// TIA Portal V15.1 export
// export: Created 2024-06-21T08:41:14.0911961Z, ExportSetting WithDefaults, DisplayName Totally Integrated Automation Portal, DisplayVersion V15.1 Update 5, DisplayName TIA Portal Openness, DisplayVersion V15.1 Update 5, DisplayName SINAMICS Startdrive Advanced, DisplayVersion V15.1, DisplayName G130, G150, S120, S150, SINAMICS MV, S210, DisplayVersion V15.1, DisplayName G110M, G120, G120C, G120D, G120P, DisplayVersion V15.1, DisplayName STEP 7 Professional, DisplayVersion V15.1 Update 5, DisplayName STEP 7 Safety, DisplayVersion V15.1, DisplayName WinCC Professional, DisplayVersion V15.1 Update 5, DisplayName SIMATIC Visualization Architect, DisplayVersion V15.1
FUNCTION_BLOCK "LGBSickDL100"   // FB6673, FBD
TITLE = LSickDL100 / LGBSickDL100
{ S7_Optimized_Access := 'TRUE' }
VERSION : 0.1
// LSickDL100 / LGBSickDL100
// stored: AutoNumber false, IsIECCheckEnabled false, IsRetainMemResEnabled false, MemoryReserve 100, SetENOAutomatically False, UDAEnableTagReadback false
   VAR_INPUT
      I_TEL_M04_Inputs { ExternalAccessible := 'False'; ExternalVisible := 'False'; ExternalWritable := 'False'} : "Sick_TEL_M04_Inputs";   // Sick input module M04
      I_TEL_M10_Inputs { ExternalAccessible := 'False'; ExternalVisible := 'False'; ExternalWritable := 'False'} : "Sick_TEL_M10_Inputs";   // Sick input module M10
      I_TEL_M13_Inputs_P1 { ExternalAccessible := 'False'; ExternalVisible := 'False'; ExternalWritable := 'False'} : "Sick_TEL_M13_Inputs_Part_1";   // Sick input module M13 part 1
      I_TEL_M13_Inputs_P2 { ExternalAccessible := 'False'; ExternalVisible := 'False'; ExternalWritable := 'False'} : "Sick_TEL_M13_Inputs_Part_2";   // Sick input module M13 part 2
      I_TurnLaserOff { ExternalAccessible := 'False'; ExternalVisible := 'False'; ExternalWritable := 'False'} : Bool;   // Turn laser off, this will cause a alarm B !
      C_ReceptionQualityMin { ExternalAccessible := 'False'; ExternalVisible := 'False'; ExternalWritable := 'False'} : Int := -96;   // Minimum reception quality level before alarm C
   END_VAR
   VAR_OUTPUT
      O_TEL_M10_Outputs { ExternalAccessible := 'False'; ExternalVisible := 'False'; ExternalWritable := 'False'} : "Sick_TEL_M10_Outputs";   // Sick output module M10
      O_Distance { ExternalAccessible := 'False'; ExternalVisible := 'False'; ExternalWritable := 'False'} : DInt;   // Current distance in the current resolution under consideration of offset. Depending on resolution, one digit corresponds to 0.1 to 100 mm.
      O_Speed { ExternalAccessible := 'False'; ExternalVisible := 'False'; ExternalWritable := 'False'} : DInt;   // Current speed in selected resolution. Depending on resolution, one digit corresponds to 0.1m/s to 100 mm/s.
      O_DeviceTemp { ExternalAccessible := 'False'; ExternalVisible := 'False'; ExternalWritable := 'False'} : SInt := 0;   // Device temperature [°C]
      O_ReceptionQuality { ExternalAccessible := 'False'; ExternalVisible := 'False'; ExternalWritable := 'False'} : Int := 0;   // Device-specific value for the signal reception quality
      O_OperatingHours { ExternalAccessible := 'False'; ExternalVisible := 'False'; ExternalWritable := 'False'} : Int := 0;   // Operating hours in 10 hour units.
      O_LaserOff { ExternalAccessible := 'False'; ExternalVisible := 'False'; ExternalWritable := 'False'} : Bool;   // Laser is off
      O_AlarmABCondition { ExternalAccessible := 'False'; ExternalVisible := 'False'; ExternalWritable := 'False'} : Bool;   // Alarm AB Condition
      O_AlarmA { ExternalAccessible := 'False'; ExternalVisible := 'False'; ExternalWritable := 'False'} : Bool;   // Alarm A
      O_AlarmB { ExternalAccessible := 'False'; ExternalVisible := 'False'; ExternalWritable := 'False'} : Bool;   // Alarm B
      O_AlarmC { ExternalAccessible := 'False'; ExternalVisible := 'False'; ExternalWritable := 'False'} : Bool;   // Alarm C
      O_AlarmD { ExternalAccessible := 'False'; ExternalVisible := 'False'; ExternalWritable := 'False'} : Bool;   // Alarm D
      H_AlarmDWord { ExternalAccessible := 'False'; ExternalVisible := 'False'; ExternalWritable := 'False'} : DWord;   // Alarm Word
   END_VAR
   VAR_IN_OUT
      IO_Modes : "Modes";   // Modes
      H_HMI : "H_HMI";   // Animation
      H_GBSickDL100 : "H_GBSickDL100";   // Animation
   END_VAR
   VAR
      AB_PlausibilityError { ExternalAccessible := 'False'; ExternalVisible := 'False'; ExternalWritable := 'False'} : Bool;   // No valid measurement value can be calculated.
      AB_TemperatureError { ExternalAccessible := 'False'; ExternalVisible := 'False'; ExternalWritable := 'False'} : Bool;   // The device is also operated outside of the specified temperature range
      AB_SignalLevelError { ExternalAccessible := 'False'; ExternalVisible := 'False'; ExternalWritable := 'False'} : Bool;   // The measured signal level is too low.
      AB_LaserError { ExternalAccessible := 'False'; ExternalVisible := 'False'; ExternalWritable := 'False'} : Bool;   // The laser may have reached the end of its service life
      AB_LaserOff { ExternalAccessible := 'False'; ExternalVisible := 'False'; ExternalWritable := 'False'} : Bool;   // Laser is off
      AB_ValueValid { ExternalAccessible := 'False'; ExternalVisible := 'False'; ExternalWritable := 'False'} : Bool;   // 1= No distance or speed measurement value can be read. 0 = Current measurement value is valid
      AC_PlausibilityWarning { ExternalAccessible := 'False'; ExternalVisible := 'False'; ExternalWritable := 'False'} : Bool;   // Measured values are impaired.
      AC_TemperatureWarning { ExternalAccessible := 'False'; ExternalVisible := 'False'; ExternalWritable := 'False'} : Bool;   // The ambient temperature is only just within the permissible range.
      AC_SignalLevelWarning { ExternalAccessible := 'False'; ExternalVisible := 'False'; ExternalWritable := 'False'} : Bool;   // The measured signal level is close to the permissible range.
      AC_LaserWarning { ExternalAccessible := 'False'; ExternalVisible := 'False'; ExternalWritable := 'False'} : Bool;   // The laser has reached its service life.
      AC_ReceptionQuality { ExternalAccessible := 'False'; ExternalVisible := 'False'; ExternalWritable := 'False'} : Bool;   // Device-specific value for the signal reception quality
      AlarmABCondition { ExternalAccessible := 'False'; ExternalVisible := 'False'; ExternalWritable := 'False'} : Bool;   // Alarm AB Condition
      AlarmA { ExternalAccessible := 'False'; ExternalVisible := 'False'; ExternalWritable := 'False'} : Bool;   // Alarm A
      AlarmB { ExternalAccessible := 'False'; ExternalVisible := 'False'; ExternalWritable := 'False'} : Bool;   // Alarm B
      AlarmC { ExternalAccessible := 'False'; ExternalVisible := 'False'; ExternalWritable := 'False'} : Bool;   // Alarm C
      AlarmD { ExternalAccessible := 'False'; ExternalVisible := 'False'; ExternalWritable := 'False'} : Bool;   // Alarm D
   END_VAR
   VAR_TEMP   // added for the SCL form of the ladder/FBD networks
      _w1 : Bool;
   END_VAR
BEGIN

REGION Network 1: **** 2.2 - Alarms - Alarm Generation **** Alarm B laser is turned off
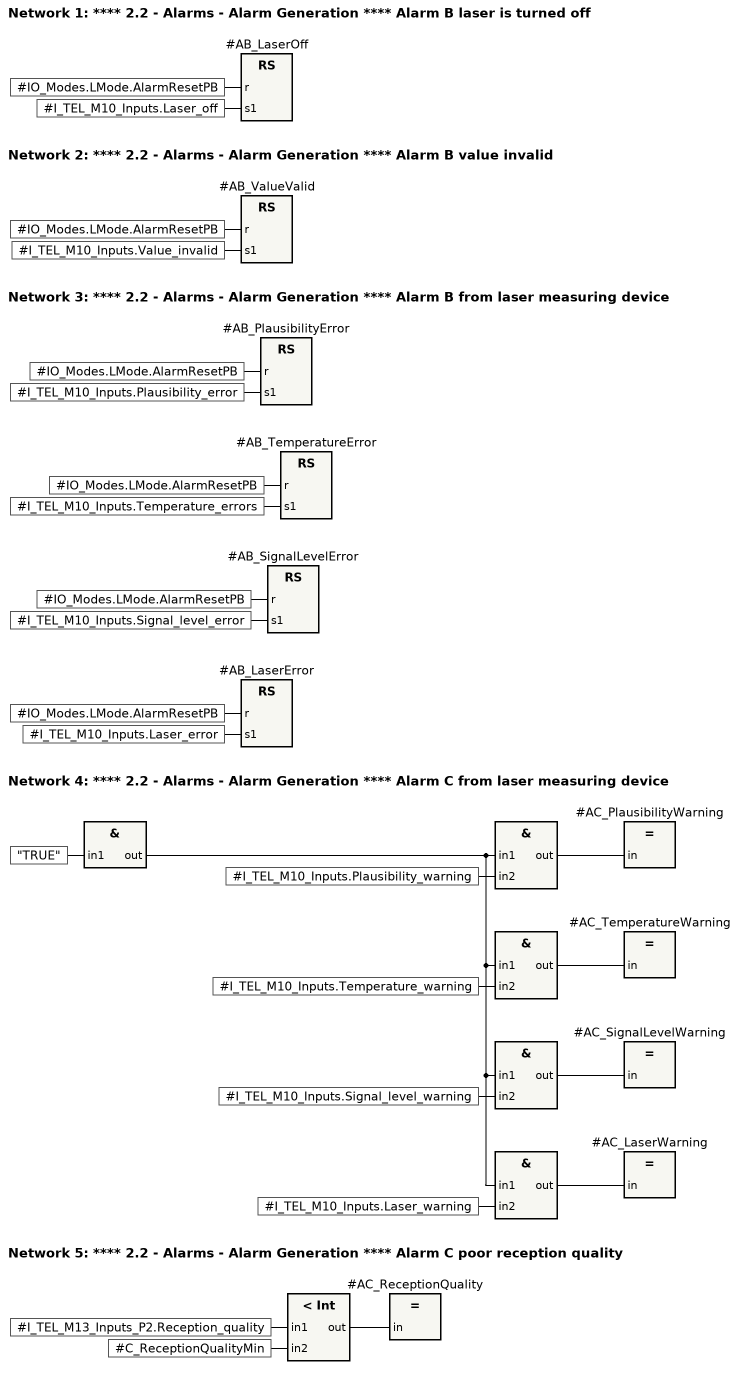
   IF #IO_Modes.LMode.AlarmResetPB THEN
       #AB_LaserOff := FALSE;   // RS flip-flop
   END_IF;
   IF #I_TEL_M10_Inputs.Laser_off THEN #AB_LaserOff := TRUE; END_IF;
END_REGION

REGION Network 2: **** 2.2 - Alarms - Alarm Generation **** Alarm B value invalid
   IF #IO_Modes.LMode.AlarmResetPB THEN
       #AB_ValueValid := FALSE;   // RS flip-flop
   END_IF;
   IF #I_TEL_M10_Inputs.Value_invalid THEN #AB_ValueValid := TRUE; END_IF;
END_REGION

REGION Network 3: **** 2.2 - Alarms - Alarm Generation **** Alarm B from laser measuring device
   IF #IO_Modes.LMode.AlarmResetPB THEN
       #AB_PlausibilityError := FALSE;   // RS flip-flop
   END_IF;
   IF #I_TEL_M10_Inputs.Plausibility_error THEN #AB_PlausibilityError := TRUE; END_IF;
   IF #IO_Modes.LMode.AlarmResetPB THEN
       #AB_TemperatureError := FALSE;   // RS flip-flop: __ 40°C l l l~l 20°C l l l l l l 0°C l l l l -10°C l l (__)
   END_IF;
   IF #I_TEL_M10_Inputs.Temperature_errors THEN #AB_TemperatureError := TRUE; END_IF;
   IF #IO_Modes.LMode.AlarmResetPB THEN
       #AB_SignalLevelError := FALSE;   // RS flip-flop
   END_IF;
   IF #I_TEL_M10_Inputs.Signal_level_error THEN #AB_SignalLevelError := TRUE; END_IF;
   IF #IO_Modes.LMode.AlarmResetPB THEN
       #AB_LaserError := FALSE;   // RS flip-flop
   END_IF;
   IF #I_TEL_M10_Inputs.Laser_error THEN #AB_LaserError := TRUE; END_IF;
END_REGION

REGION Network 4: **** 2.2 - Alarms - Alarm Generation **** Alarm C from laser measuring device
   #AC_PlausibilityWarning := "TRUE" AND #I_TEL_M10_Inputs.Plausibility_warning;
   #AC_TemperatureWarning := "TRUE" AND #I_TEL_M10_Inputs.Temperature_warning;   // __ 40°C l l l~l 20°C l l l l l l 0°C l l l l -10°C l l (__)
   #AC_SignalLevelWarning := "TRUE" AND #I_TEL_M10_Inputs.Signal_level_warning;
   #AC_LaserWarning := "TRUE" AND #I_TEL_M10_Inputs.Laser_warning;
END_REGION

REGION Network 5: **** 2.2 - Alarms - Alarm Generation **** Alarm C poor reception quality
   #AC_ReceptionQuality := #I_TEL_M13_Inputs_P2.Reception_quality < #C_ReceptionQualityMin;   // ^ Reception quality (%) l -32db l_______________ l \ OK area min. l \ if quality drops below this level .setting l---------------------------------------\------------------------------------------------------------- an alarm C is created. l \ alarm C area -96db l________________________\___________________________> Time (h) l This can be caused: -by dirt on the mirror. -misalignment (ex. cuased by moving the mirror). -...
END_REGION

REGION Network 6: **** 4.6 - Machine Status - Indication **** Icon Animation
   // Icon Animation
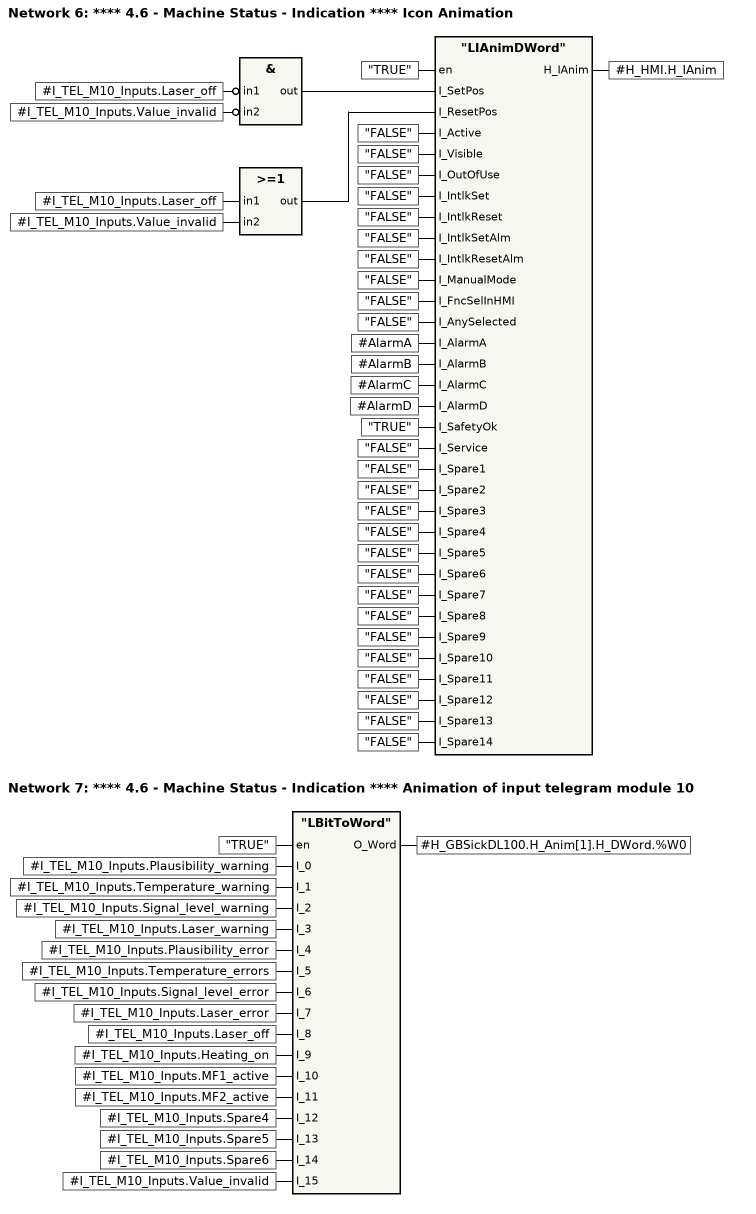
   IF "TRUE" THEN
       "LIAnimDWord"(I_SetPos := NOT #I_TEL_M10_Inputs.Laser_off AND NOT #I_TEL_M10_Inputs.Value_invalid,   // HMI PLC __________________________________________________________ l _SIEMENS____________________________SIMATIC HMI_____ l ___________________ l l l l l_l_l_l______________l l l l l l SIEMENS SIMATIC l l l l l l ________S7-1500 l l l l l l l___________O_l l l l Icon l l l l l l l l ____ l l l l l l l l l l l l l l l l l l l____l <<-------==================l= l========= l l l l l l l l l l______________l l l l IAnim l l l ___ l l l l l l __l l__ l l l l l l l__ __l l l l l l l l___l l l l l l l l l l_____________________________________________________ l l l__________________ l l_________________________________________________________ l Icon animation word is send to the HMI to be used in ex .modezone screen _
                     I_ResetPos := #I_TEL_M10_Inputs.Laser_off OR #I_TEL_M10_Inputs.Value_invalid,
                     I_Active := "FALSE",
                     I_Visible := "FALSE",
                     I_OutOfUse := "FALSE",
                     I_IntlkSet := "FALSE",
                     I_IntlkReset := "FALSE",
                     I_IntlkSetAlm := "FALSE",
                     I_IntlkResetAlm := "FALSE",
                     I_ManualMode := "FALSE",
                     I_FncSelInHMI := "FALSE",
                     I_AnySelected := "FALSE",
                     I_AlarmA := #AlarmA,
                     I_AlarmB := #AlarmB,
                     I_AlarmC := #AlarmC,
                     I_AlarmD := #AlarmD,
                     I_SafetyOk := "TRUE",
                     I_Service := "FALSE",
                     I_Spare1 := "FALSE",
                     I_Spare2 := "FALSE",
                     I_Spare3 := "FALSE",
                     I_Spare4 := "FALSE",
                     I_Spare5 := "FALSE",
                     I_Spare6 := "FALSE",
                     I_Spare7 := "FALSE",
                     I_Spare8 := "FALSE",
                     I_Spare9 := "FALSE",
                     I_Spare10 := "FALSE",
                     I_Spare11 := "FALSE",
                     I_Spare12 := "FALSE",
                     I_Spare13 := "FALSE",
                     I_Spare14 := "FALSE",
                     H_IAnim => #H_HMI.H_IAnim);
   END_IF;
END_REGION

REGION Network 7: **** 4.6 - Machine Status - Indication **** Animation of input telegram module 10
   // Animation
   IF "TRUE" THEN
       "LBitToWord"(I_0 := #I_TEL_M10_Inputs.Plausibility_warning,   // HMI PLC __________________________________________________________ l _SIEMENS____________________________SIMATIC HMI_____ l ___________________ l l l l l_l_l_l______________l l l l l l SIEMENS SIMATIC l l l ________________ l l l ________S7-1500 l l l l_____________ X l l l l l___________O_l l l l l l l l l l l l l l l Popup or l l l l l l l l l l screen. l l l l l l l l l l l <<-------==================l= l========= l l l l l l l Anim l l l l l______________l l l l l_______________l l l l ___ l l l l l l __l l__ l l l l l l l__ __l l l l l l l l___l l l l l l l l l l_____________________________________________________ l l l__________________ l l_________________________________________________________ l Animation word is send to the HMI to be used in object screen or popup _
                    I_1 := #I_TEL_M10_Inputs.Temperature_warning,
                    I_2 := #I_TEL_M10_Inputs.Signal_level_warning,
                    I_3 := #I_TEL_M10_Inputs.Laser_warning,
                    I_4 := #I_TEL_M10_Inputs.Plausibility_error,
                    I_5 := #I_TEL_M10_Inputs.Temperature_errors,
                    I_6 := #I_TEL_M10_Inputs.Signal_level_error,
                    I_7 := #I_TEL_M10_Inputs.Laser_error,
                    I_8 := #I_TEL_M10_Inputs.Laser_off,
                    I_9 := #I_TEL_M10_Inputs.Heating_on,
                    I_10 := #I_TEL_M10_Inputs.MF1_active,
                    I_11 := #I_TEL_M10_Inputs.MF2_active,
                    I_12 := #I_TEL_M10_Inputs.Spare4,
                    I_13 := #I_TEL_M10_Inputs.Spare5,
                    I_14 := #I_TEL_M10_Inputs.Spare6,
                    I_15 := #I_TEL_M10_Inputs.Value_invalid,
                    O_Word => #H_GBSickDL100.H_Anim[1].H_DWord.%W0);
   END_IF;
END_REGION

REGION Network 8: **** 4.6 - Machine Status - Indication **** Animation of output telegram module 10
   // Animation
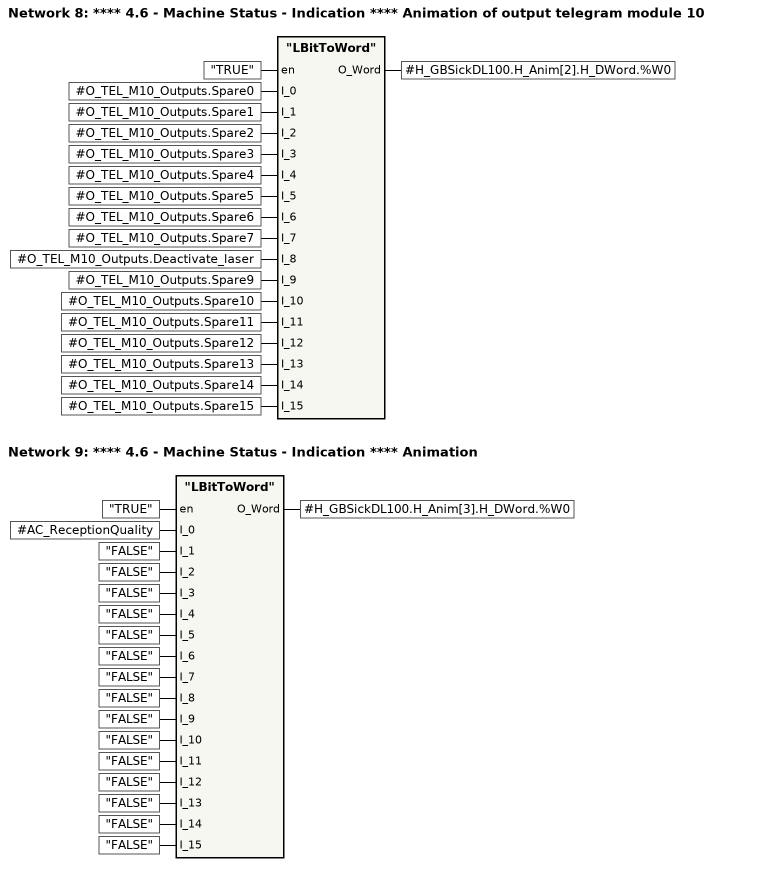
   IF "TRUE" THEN
       "LBitToWord"(I_0 := #O_TEL_M10_Outputs.Spare0,   // HMI PLC __________________________________________________________ l _SIEMENS____________________________SIMATIC HMI_____ l ___________________ l l l l l_l_l_l______________l l l l l l SIEMENS SIMATIC l l l ________________ l l l ________S7-1500 l l l l_____________ X l l l l l___________O_l l l l l l l l l l l l l l l Popup or l l l l l l l l l l screen. l l l l l l l l l l l <<-------==================l= l========= l l l l l l l Anim l l l l l______________l l l l l_______________l l l l ___ l l l l l l __l l__ l l l l l l l__ __l l l l l l l l___l l l l l l l l l l_____________________________________________________ l l l__________________ l l_________________________________________________________ l Animation word is send to the HMI to be used in object screen or popup _
                    I_1 := #O_TEL_M10_Outputs.Spare1,
                    I_2 := #O_TEL_M10_Outputs.Spare2,
                    I_3 := #O_TEL_M10_Outputs.Spare3,
                    I_4 := #O_TEL_M10_Outputs.Spare4,
                    I_5 := #O_TEL_M10_Outputs.Spare5,
                    I_6 := #O_TEL_M10_Outputs.Spare6,
                    I_7 := #O_TEL_M10_Outputs.Spare7,
                    I_8 := #O_TEL_M10_Outputs.Deactivate_laser,
                    I_9 := #O_TEL_M10_Outputs.Spare9,
                    I_10 := #O_TEL_M10_Outputs.Spare10,
                    I_11 := #O_TEL_M10_Outputs.Spare11,
                    I_12 := #O_TEL_M10_Outputs.Spare12,
                    I_13 := #O_TEL_M10_Outputs.Spare13,
                    I_14 := #O_TEL_M10_Outputs.Spare14,
                    I_15 := #O_TEL_M10_Outputs.Spare15,
                    O_Word => #H_GBSickDL100.H_Anim[2].H_DWord.%W0);
   END_IF;
END_REGION

REGION Network 9: **** 4.6 - Machine Status - Indication **** Animation
   // Animation
   IF "TRUE" THEN
       "LBitToWord"(I_0 := #AC_ReceptionQuality,   // HMI PLC __________________________________________________________ l _SIEMENS____________________________SIMATIC HMI_____ l ___________________ l l l l l_l_l_l______________l l l l l l SIEMENS SIMATIC l l l ________________ l l l ________S7-1500 l l l l_____________ X l l l l l___________O_l l l l l l l l l l l l l l l Popup or l l l l l l l l l l screen. l l l l l l l l l l l <<-------==================l= l========= l l l l l l l Anim l l l l l______________l l l l l_______________l l l l ___ l l l l l l __l l__ l l l l l l l__ __l l l l l l l l___l l l l l l l l l l_____________________________________________________ l l l__________________ l l_________________________________________________________ l Animation word is send to the HMI to be used in object screen or popup _
                    I_1 := "FALSE",
                    I_2 := "FALSE",
                    I_3 := "FALSE",
                    I_4 := "FALSE",
                    I_5 := "FALSE",
                    I_6 := "FALSE",
                    I_7 := "FALSE",
                    I_8 := "FALSE",
                    I_9 := "FALSE",
                    I_10 := "FALSE",
                    I_11 := "FALSE",
                    I_12 := "FALSE",
                    I_13 := "FALSE",
                    I_14 := "FALSE",
                    I_15 := "FALSE",
                    O_Word => #H_GBSickDL100.H_Anim[3].H_DWord.%W0);
   END_IF;
END_REGION

REGION Network 10: **** 4.6 - Machine Status - Indication **** Animation
   // Animation
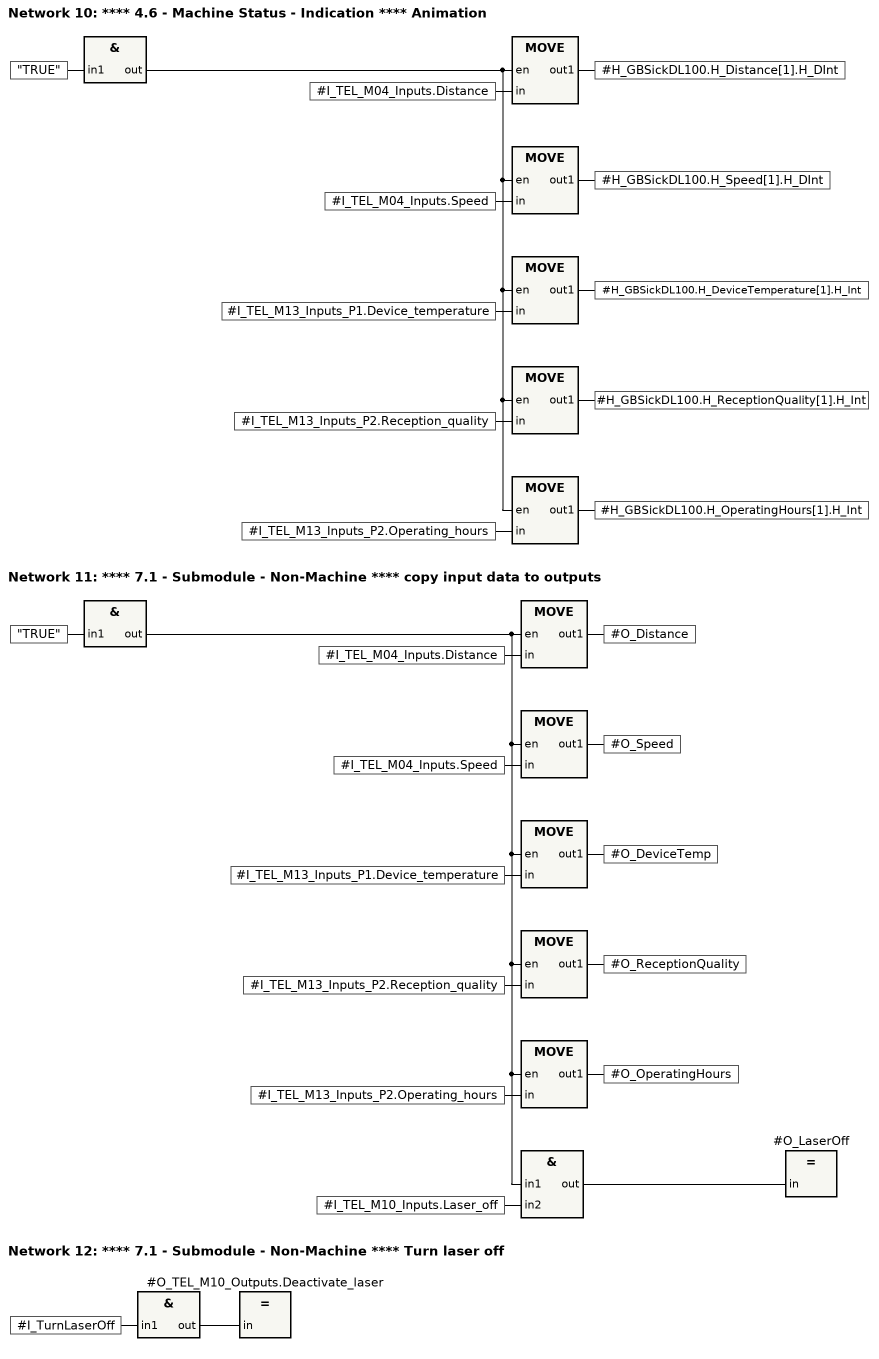
   IF "TRUE" THEN
       #H_GBSickDL100.H_Distance[1].H_DInt := #I_TEL_M04_Inputs.Distance;   // HMI PLC __________________________________________________________ l _SIEMENS____________________________SIMATIC HMI_____ l ___________________ l l l l l_l_l_l______________l l l l l l SIEMENS SIMATIC l l l ________________ l l l ________S7-1500 l l l l_____________ X l l l l l___________O_l l l l l l l l l l l l l l l Popup or l l l l l l l l l l screen. l l l l l l l l l l l <<-------==================l= l========= l l l l l l l Anim l l l l l______________l l l l l_______________l l l l ___ l l l l l l __l l__ l l l l l l l__ __l l l l l l l l___l l l l l l l l l l_____________________________________________________ l l l__________________ l l_________________________________________________________ l Animation word is send to the HMI to be used in object screen or popup _
       #H_GBSickDL100.H_Speed[1].H_DInt := #I_TEL_M04_Inputs.Speed;
       #H_GBSickDL100.H_DeviceTemperature[1].H_Int := #I_TEL_M13_Inputs_P1.Device_temperature;
       #H_GBSickDL100.H_ReceptionQuality[1].H_Int := #I_TEL_M13_Inputs_P2.Reception_quality;
       #H_GBSickDL100.H_OperatingHours[1].H_Int := #I_TEL_M13_Inputs_P2.Operating_hours;
   END_IF;
END_REGION

REGION Network 11: **** 7.1 - Submodule - Non-Machine **** copy input data to outputs
   IF "TRUE" THEN
       #O_Distance := #I_TEL_M04_Inputs.Distance;
       #O_Speed := #I_TEL_M04_Inputs.Speed;
       #O_DeviceTemp := #I_TEL_M13_Inputs_P1.Device_temperature;
       #O_ReceptionQuality := #I_TEL_M13_Inputs_P2.Reception_quality;
       #O_OperatingHours := #I_TEL_M13_Inputs_P2.Operating_hours;
   END_IF;
   #O_LaserOff := "TRUE" AND #I_TEL_M10_Inputs.Laser_off;   // _____ l \ l / l // l< l ---O-- l--------------------//------------------------- l< l_ / l \_l // l< l l ON state ****************************** _____ OFF state l \ l / l l< l ---O-- l l< l_ / l \_l l< l l _
END_REGION

REGION Network 12: **** 7.1 - Submodule - Non-Machine **** Turn laser off
   #O_TEL_M10_Outputs.Deactivate_laser := #I_TurnLaserOff;   // _____ l \ l / l // l< l ---O-- l--------------------//------------------------- l< l_ / l \_l // l< l l ON state ****************************** _____ OFF state l \ l / l l< l ---O-- l l< l_ / l \_l l< l l _
END_REGION

REGION Network 13: **** 9 - Alarm Summary **** Alarm A
   // Alarm A
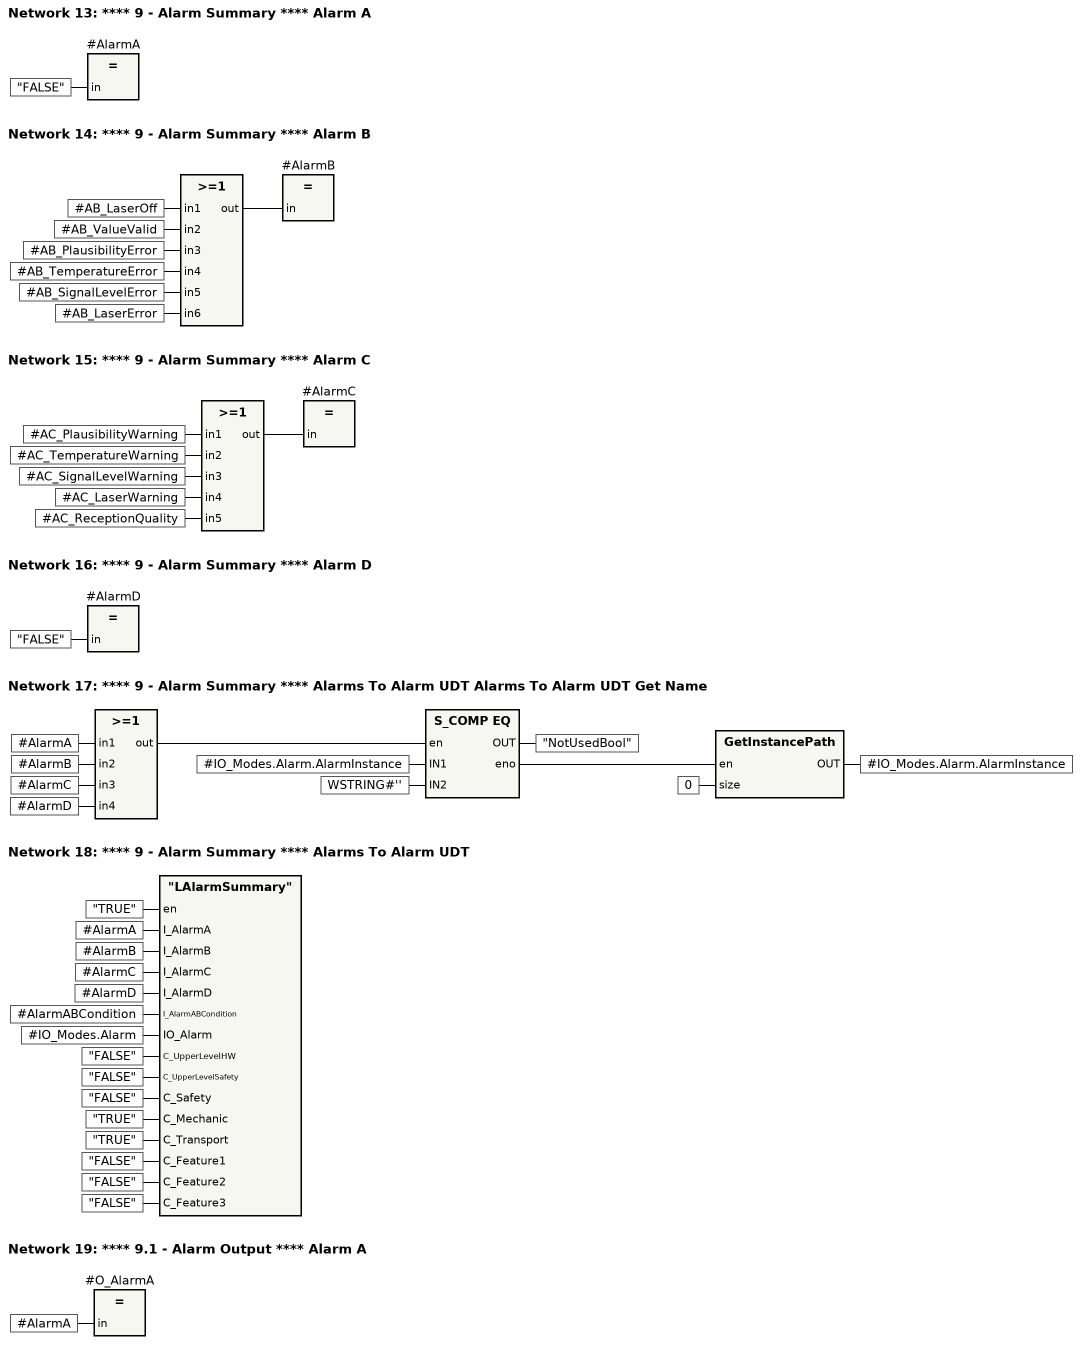
   #AlarmA := "FALSE";
END_REGION

REGION Network 14: **** 9 - Alarm Summary **** Alarm B
   // Alarm B
   #AlarmB := #AB_LaserOff OR #AB_ValueValid OR #AB_PlausibilityError OR #AB_TemperatureError OR #AB_SignalLevelError OR #AB_LaserError;
END_REGION

REGION Network 15: **** 9 - Alarm Summary **** Alarm C
   // Alarm C
   #AlarmC := #AC_PlausibilityWarning OR #AC_TemperatureWarning OR #AC_SignalLevelWarning OR #AC_LaserWarning OR #AC_ReceptionQuality;
END_REGION

REGION Network 16: **** 9 - Alarm Summary **** Alarm D
   // Alarm D
   #AlarmD := "FALSE";
END_REGION

REGION Network 17: **** 9 - Alarm Summary **** Alarms To Alarm UDT Alarms To Alarm UDT Get Name
   // Alarms To Alarm UDT Alarms To Alarm UDT Get Name
   S_COMP(EN := #AlarmA OR #AlarmB OR #AlarmC OR #AlarmD,
          IN1 := #IO_Modes.Alarm.AlarmInstance,
          IN2 := WSTRING#'',
          OUT => "NotUsedBool",
          ENO => #_w1);
   IF #_w1 THEN GetInstancePath(size := 0, OUT => #IO_Modes.Alarm.AlarmInstance); END_IF;
END_REGION

REGION Network 18: **** 9 - Alarm Summary **** Alarms To Alarm UDT
   // Alarms To Alarm UDT
   IF "TRUE" THEN
       "LAlarmSummary"(I_AlarmA := #AlarmA,
                       I_AlarmB := #AlarmB,
                       I_AlarmC := #AlarmC,
                       I_AlarmD := #AlarmD,
                       I_AlarmABCondition := #AlarmABCondition,
                       IO_Alarm := #IO_Modes.Alarm,
                       C_UpperLevelHW := "FALSE",
                       C_UpperLevelSafety := "FALSE",
                       C_Safety := "FALSE",
                       C_Mechanic := "TRUE",
                       C_Transport := "TRUE",
                       C_Feature1 := "FALSE",
                       C_Feature2 := "FALSE",
                       C_Feature3 := "FALSE");
   END_IF;
END_REGION

REGION Network 19: **** 9.1 - Alarm Output **** Alarm A
   // Alarm A
   #O_AlarmA := #AlarmA;
END_REGION

REGION Network 20: **** 9.1 - Alarm Output **** Alarm B
   // Alarm B
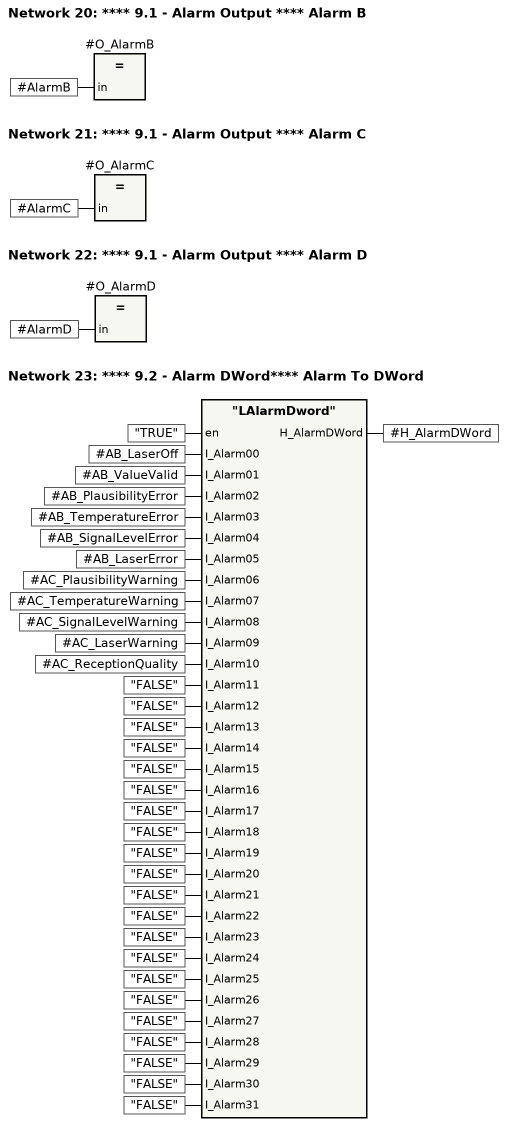
   #O_AlarmB := #AlarmB;
END_REGION

REGION Network 21: **** 9.1 - Alarm Output **** Alarm C
   // Alarm C
   #O_AlarmC := #AlarmC;
END_REGION

REGION Network 22: **** 9.1 - Alarm Output **** Alarm D
   // Alarm D
   #O_AlarmD := #AlarmD;
END_REGION

REGION Network 23: **** 9.2 - Alarm DWord**** Alarm To DWord
   // Alarm To Word
   IF "TRUE" THEN
       "LAlarmDword"(I_Alarm00 := #AB_LaserOff,   // 1) Collets all alarms in a alarm DB through DWords ______________ ______________ l FB l l DB l l l l Current cycle l l l l l l l l l l AlarmDWord l-- =====> l l l______________l l______________l 2) Compare DB's to check for new alarms ex. DB30 ex. DB130 ______________ ______________ l DB l l DB l l Current cycle l l Previous cycle l l l Compare l l l l l l l l l l l______________l l______________l 3) Generate an alarm message on HMI (alarms linking need to be generated with TIA openess script) HMI PLC __________________________________________________________ l _SIEMENS____________________________SIMATIC HMI_____ l ___________________ l l ex. _000Passivation.AA_F00200 | A | I/O Passivation l l l_l_l_l______________l l l_____________________________________________________ l l l SIEMENS SIMATIC l l l l l l ________S7-1500 l l l l l l l___________O_l l l l l l l l l l l l l l l l l l l l DB30, DB31, DB32, ... l l l l l l l l <<-------==================l= l========= l l l l l l l l l l______________l l l l l l l ___ l l l l l l __l l__ l l l l l l l__ __l l l l l l l l___l l l l l l l l l l_____________________________________________________ l l l__________________ l l_________________________________________________________ l _
                     I_Alarm01 := #AB_ValueValid,
                     I_Alarm02 := #AB_PlausibilityError,
                     I_Alarm03 := #AB_TemperatureError,
                     I_Alarm04 := #AB_SignalLevelError,
                     I_Alarm05 := #AB_LaserError,
                     I_Alarm06 := #AC_PlausibilityWarning,
                     I_Alarm07 := #AC_TemperatureWarning,
                     I_Alarm08 := #AC_SignalLevelWarning,
                     I_Alarm09 := #AC_LaserWarning,
                     I_Alarm10 := #AC_ReceptionQuality,
                     I_Alarm11 := "FALSE",
                     I_Alarm12 := "FALSE",
                     I_Alarm13 := "FALSE",
                     I_Alarm14 := "FALSE",
                     I_Alarm15 := "FALSE",
                     I_Alarm16 := "FALSE",
                     I_Alarm17 := "FALSE",
                     I_Alarm18 := "FALSE",
                     I_Alarm19 := "FALSE",
                     I_Alarm20 := "FALSE",
                     I_Alarm21 := "FALSE",
                     I_Alarm22 := "FALSE",
                     I_Alarm23 := "FALSE",
                     I_Alarm24 := "FALSE",
                     I_Alarm25 := "FALSE",
                     I_Alarm26 := "FALSE",
                     I_Alarm27 := "FALSE",
                     I_Alarm28 := "FALSE",
                     I_Alarm29 := "FALSE",
                     I_Alarm30 := "FALSE",
                     I_Alarm31 := "FALSE",
                     H_AlarmDWord => #H_AlarmDWord);
   END_IF;
END_REGION
END_FUNCTION_BLOCK
